FUNCTION_BLOCK ABSTRACT FB_SimStation IMPLEMENTS IStation
VAR_INPUT
END_VAR
VAR_OUTPUT
END_VAR
VAR
	bPartPresent				AT %I* : BOOL;
	bReady						: BOOL;
	bFaulted					: BOOL;
	
	StationState				: E_SimStationState;
	pPartStatus					: POINTER TO ST_PartStatus;
	tmrDelay					: TON;
END_VAR

METHOD PROTECTED ABSTRACT DoWork : BOOL
VAR_INPUT
END_VAR
END_METHOD

METHOD Execute : PVOID
CASE StationState OF
	
	E_SimStationState.IDLE:
		
		tmrDelay(IN:=bPartPresent, PT:=T#100MS);
		
		IF bPartPresent THEN
			bReady := FALSE;
			IF tmrDelay.Q THEN
				StationState := E_SimStationState.WORKING;
			END_IF
		ELSE
			bReady := TRUE;
		END_IF
		
	E_SimStationState.WORKING:
		
		bReady := FALSE;
		
		IF DoWork() THEN
			StationState := E_SimStationState.DONE;
		END_IF
	
	E_SimStationState.DONE:
	
		bReady := TRUE;
		
		IF NOT bPartPresent THEN
			UpdatePartStatus();
			StationState := E_SimStationState.IDLE;
		END_IF
		
END_CASE
END_METHOD

PROPERTY Faulted : BOOL
GET
Faulted := bFaulted;
END_GET
END_PROPERTY

PROPERTY PartPresent : BOOL
GET
PartPresent := bPartPresent;
END_GET
END_PROPERTY

PROPERTY PartStatus : POINTER TO ST_PartStatus
SET
pPartStatus := PartStatus;
END_SET
END_PROPERTY

PROPERTY Ready : BOOL
GET
Ready := bReady;
END_GET
END_PROPERTY

METHOD PROTECTED ABSTRACT UpdatePartStatus : PVOID
VAR_INPUT
END_VAR
END_METHOD

END_FUNCTION_BLOCK

(* stored: Version 1.1.0.1, ProductVersion 3.1.4024.12
   POU FB_SimStation: Id {652e3183-24a4-44ce-821b-86424bd43b56}, SpecialFunc None
   Method DoWork: Id {ecc776db-db39-47b6-ab26-9a292e8a2694}
   Method Execute: Id {810bc9a2-3455-4001-b511-f17f596081c2}
   Property Faulted: Id {08a80eca-2fd7-4430-8828-a9e5b69b7479}
   Get Get: Id {0c0f5e8e-2d04-4c34-9a2e-9fb3de86cf0d}
   Property PartPresent: Id {b8cf2840-06cb-4324-b340-2bd471b18987}
   Get Get: Id {6c61540d-d53c-4f21-a792-f4070c5aac11}
   Property PartStatus: Id {1e680408-f976-40e4-9e94-be3fe2c6fcdb}
   Set Set: Id {525e35f7-1820-415a-9700-c5d36d610128}
   Property Ready: Id {01c818ef-b4cd-457f-8d89-c6695942a95b}
   Get Get: Id {064696c7-b595-402f-8346-af9fef0ba8c6}
   Method UpdatePartStatus: Id {1931ee90-b418-424e-b0a8-d3a0a0a746a0} *)
